TYPE ST_Chamber1_Signal_In :
STRUCT
	bDoorClosed : BOOL;
	rTemperature : REAL;

	bDIs : ARRAY[1..16] OF BOOL;
	rAIs : ARRAY[1..16] OF REAL;
END_STRUCT
END_TYPE

(* stored: Version 1.1.0.1, ProductVersion 3.1.4026.18
   DUT ST_Chamber1_Signal_In: Id {01a04f04-4882-4cc0-9760-4299fa29ec69} *)
